// TIA Portal V18 export
// export: Created 2026-06-08T16:32:20.8214944Z, ExportSetting WithDefaults, DisplayName Totally Integrated Automation Portal, DisplayVersion V18, DisplayName TIA Portal Openness, DisplayVersion V18, DisplayName TIA Portal Version Control Interface, DisplayVersion V18, DisplayName STEP 7 Professional, DisplayVersion V18, DisplayName STEP 7 Safety, DisplayVersion V18, DisplayName WinCC Professional, DisplayVersion V18
FUNCTION_BLOCK "base_production_fb"   // FB5, LAD
VERSION : 0.1
// stored: AutoNumber true, IsIECCheckEnabled false, UDAEnableTagReadback false
BEGIN

REGION Network 1: base_production_station
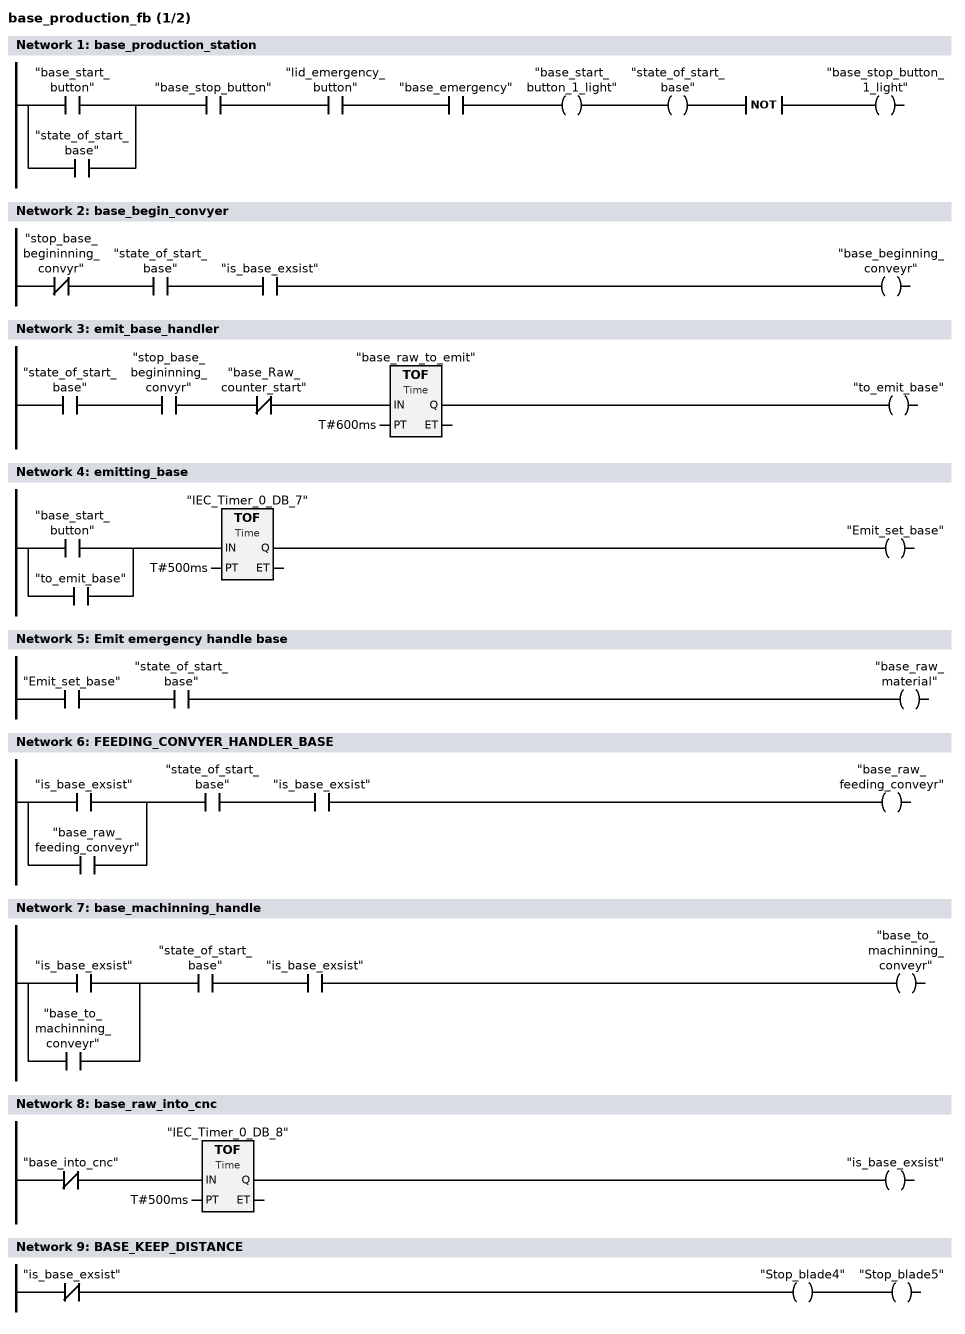
   RUNG wire#powerrail
      Contact( "base_start_button" )
      wire#w1
      Contact( "base_stop_button" )
      Contact( "lid_emergency_button" )
      Contact( "base_emergency" )
      Coil( "base_start_button_1_light" )
      Coil( "state_of_start_base" )
      Not()
      Coil( "base_stop_button_1_light" )
   END_RUNG
   RUNG wire#powerrail
      Contact( "state_of_start_base" )
   END_RUNG wire#w1
   // the same network as SCL:
   "base_start_button_1_light" := ("base_start_button" OR "state_of_start_base") AND "base_stop_button" AND "lid_emergency_button" AND "base_emergency";
   "state_of_start_base" := "base_start_button_1_light";
   "base_stop_button_1_light" := NOT "base_start_button_1_light";
END_REGION

REGION Network 2: base_begin_convyer
   RUNG wire#powerrail
      I_Contact( "stop_base_begininning_convyr" )
      Contact( "state_of_start_base" )
      Contact( "is_base_exsist" )
      Coil( "base_beginning_conveyr" )
   END_RUNG
   // the same network as SCL:
   "base_beginning_conveyr" := NOT "stop_base_begininning_convyr" AND "state_of_start_base" AND "is_base_exsist";
END_REGION

REGION Network 3: emit_base_handler
   RUNG wire#powerrail
      Contact( "state_of_start_base" )
      Contact( "stop_base_begininning_convyr" )
      I_Contact( "base_Raw_counter_start" )
      { S7_Templates := "time_type := Time" } "base_raw_to_emit".TOF(pt := T#600ms, et =>)
      Coil( "to_emit_base" )
   END_RUNG
   // the same network as SCL:
   "base_raw_to_emit".TOF(IN := "state_of_start_base" AND "stop_base_begininning_convyr" AND NOT "base_Raw_counter_start",
                          PT := T#600ms);
   "to_emit_base" := "base_raw_to_emit".Q;
END_REGION

REGION Network 4: emitting_base
   RUNG wire#powerrail
      Contact( "base_start_button" )
      wire#w1
      { S7_Templates := "time_type := Time" } "IEC_Timer_0_DB_7".TOF(pt := T#500ms, et =>)
      Coil( "Emit_set_base" )
   END_RUNG
   RUNG wire#powerrail
      Contact( "to_emit_base" )
   END_RUNG wire#w1
   // the same network as SCL:
   "IEC_Timer_0_DB_7".TOF(IN := "base_start_button" OR "to_emit_base", PT := T#500ms);
   "Emit_set_base" := "IEC_Timer_0_DB_7".Q;
END_REGION

REGION Network 5: Emit emergency handle base
   RUNG wire#powerrail
      Contact( "Emit_set_base" )
      Contact( "state_of_start_base" )
      Coil( "base_raw_material" )
   END_RUNG
   // the same network as SCL:
   "base_raw_material" := "Emit_set_base" AND "state_of_start_base";
END_REGION

REGION Network 6: FEEDING_CONVYER_HANDLER_BASE
   RUNG wire#powerrail
      Contact( "is_base_exsist" )
      wire#w1
      Contact( "state_of_start_base" )
      Contact( "is_base_exsist" )
      Coil( "base_raw_feeding_conveyr" )
   END_RUNG
   RUNG wire#powerrail
      Contact( "base_raw_feeding_conveyr" )
   END_RUNG wire#w1
   // the same network as SCL:
   "base_raw_feeding_conveyr" := ("is_base_exsist" OR "base_raw_feeding_conveyr") AND "state_of_start_base" AND "is_base_exsist";
END_REGION

REGION Network 7: base_machinning_handle
   RUNG wire#powerrail
      Contact( "is_base_exsist" )
      wire#w1
      Contact( "state_of_start_base" )
      Contact( "is_base_exsist" )
      Coil( "base_to_machinning_conveyr" )
   END_RUNG
   RUNG wire#powerrail
      Contact( "base_to_machinning_conveyr" )
   END_RUNG wire#w1
   // the same network as SCL:
   "base_to_machinning_conveyr" := ("is_base_exsist" OR "base_to_machinning_conveyr") AND "state_of_start_base" AND "is_base_exsist";
END_REGION

REGION Network 8: base_raw_into_cnc
   RUNG wire#powerrail
      I_Contact( "base_into_cnc" )
      { S7_Templates := "time_type := Time" } "IEC_Timer_0_DB_8".TOF(pt := T#500ms, et =>)
      Coil( "is_base_exsist" )
   END_RUNG
   // the same network as SCL:
   "IEC_Timer_0_DB_8".TOF(IN := NOT "base_into_cnc", PT := T#500ms);
   "is_base_exsist" := "IEC_Timer_0_DB_8".Q;
END_REGION

REGION Network 9: BASE_KEEP_DISTANCE
   RUNG wire#powerrail
      I_Contact( "is_base_exsist" )
      Coil( "Stop_blade4" )
      Coil( "Stop_blade5" )
   END_RUNG
   // the same network as SCL:
   "Stop_blade4" := NOT "is_base_exsist";
   "Stop_blade5" := NOT "is_base_exsist";
END_REGION

REGION Network 10: base_excess
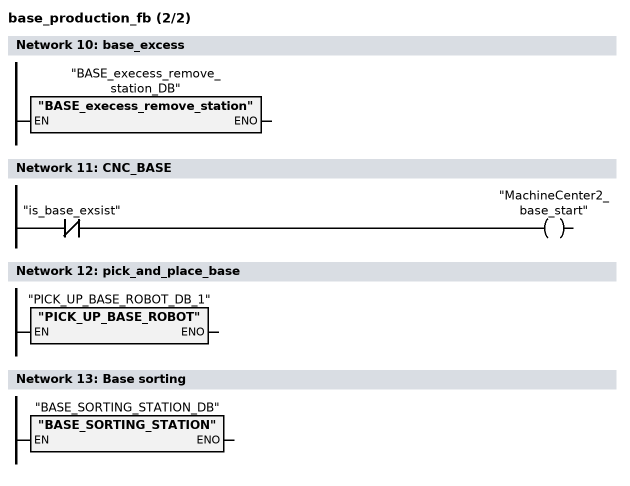
   RUNG wire#powerrail
      "BASE_execess_remove_station_DB"()
   END_RUNG
   // the same network as SCL:
   "BASE_execess_remove_station_DB"();   // "BASE_execess_remove_station"
END_REGION

REGION Network 11: CNC_BASE
   RUNG wire#powerrail
      I_Contact( "is_base_exsist" )
      Coil( "MachineCenter2_base_start" )
   END_RUNG
   // the same network as SCL:
   "MachineCenter2_base_start" := NOT "is_base_exsist";
END_REGION

REGION Network 12: pick_and_place_base
   RUNG wire#powerrail
      "PICK_UP_BASE_ROBOT_DB_1"()
   END_RUNG
   // the same network as SCL:
   "PICK_UP_BASE_ROBOT_DB_1"();   // "PICK_UP_BASE_ROBOT"
END_REGION

REGION Network 13: Base sorting
   RUNG wire#powerrail
      "BASE_SORTING_STATION_DB"()
   END_RUNG
   // the same network as SCL:
   "BASE_SORTING_STATION_DB"();   // "BASE_SORTING_STATION"
END_REGION
END_FUNCTION_BLOCK
